// TwinCAT 3 PLC project PIDtanklevel
// ProgramVersion: 3.1.4024.12
// libraries:
//   Tc2_ControllerToolbox, * (Beckhoff Automation GmbH)
//   Tc2_ModbusSrv, * (Beckhoff Automation GmbH)
//   Tc2_Standard, * (Beckhoff Automation GmbH)
//   Tc2_System, * (Beckhoff Automation GmbH)
//   Tc3_Module, * (Beckhoff Automation GmbH)
// project tree:
//   GVLs/ GlobalTags.TcGVL, InputOutputArea.TcGVL
//   / PlcTask.TcTTO
//   POUs/ ElectricBox.TcPOU, InputOutputConvert.TcPOU, MAIN.TcPOU, ModbusRead.TcPOU, ModbusWrite.TcPOU, PID.TcPOU

CONFIGURATION PIDtanklevel
    RESOURCE PLC ON TwinCAT3
        TASK PlcTask(INTERVAL := T#10ms, PRIORITY := 20);
        PROGRAM MAIN WITH PlcTask : MAIN;
    END_RESOURCE
END_CONFIGURATION

// ---- GVLs/GlobalTags.TcGVL
VAR_GLOBAL
	//
	Start 			: BOOL;
	Reset 			: BOOL;
	Stop  			: BOOL;
	//
	StartLight		: BOOL;
	ResetLight		: BOOL;
	StopLight		: BOOL;
	//
	LevelMeter 		: INT;
	FlowMeter		: INT;
	SetPoint		: INT;
	//
	FillValve		: INT;
	DischargeValve	: INT;
	SP				: INT;
	PV				: INT;
	//
	SystemStarted	: BOOL;
END_VAR

// ---- GVLs/InputOutputArea.TcGVL
VAR_GLOBAL
	InputBitArea 		: ARRAY[0..1] OF BYTE;
	OutputBitArea 		: ARRAY[0..1] OF BYTE;
	
	InputWordArea		: ARRAY[0..2] OF WORD;
	OutputWordArea		: ARRAY[0..3] OF WORD;
END_VAR

// ---- POUs/MAIN.TcPOU
PROGRAM MAIN
VAR
	InputOutputConvert: InputOutputConvert;
	PID: PID;
	ElectricBox: ElectricBox;
END_VAR

ModbusRead();
ModbusWrite();
InputOutputConvert();
PID();
ElectricBox();

END_PROGRAM

// ---- POUs/InputOutputConvert.TcPOU
FUNCTION_BLOCK InputOutputConvert
VAR_INPUT
END_VAR
VAR_OUTPUT
END_VAR
VAR
END_VAR


//Inputs
LevelMeter := (WORD_TO_INT(InputWordArea[0])*300)/1000;
FlowMeter  := (WORD_TO_INT(InputWordArea[1])*300)/1000;
SetPoint   := (WORD_TO_INT(InputWordArea[2])*300)/1000;
//Outputs
OutputWordArea[0] := INT_TO_WORD(FillValve);
OutputWordArea[1] := INT_TO_WORD(DischargeValve);
SP		   := SetPoint;
OutputWordArea[2] := INT_TO_WORD(SP);
PV		   := LevelMeter;
OutputWordArea[3] := INT_TO_WORD(PV);

//
Start := InputBitArea[0].0;
Reset := InputBitArea[0].1;
Stop  := InputBitArea[0].2;
//
OutputBitArea[0].0 := StartLight;
OutputBitArea[0].1 := ResetLight;
OutputBitArea[0].2 := StopLight;

END_FUNCTION_BLOCK

// ---- POUs/PID.TcPOU
FUNCTION_BLOCK PID
VAR_INPUT
END_VAR
VAR_OUTPUT
END_VAR
VAR
	FB_CTRL_PID: FB_CTRL_PID;
	stCTRL_PID_PARAMS: ST_CTRL_PID_PARAMS;
	Init : BOOL:=TRUE;
	fManSyncValue : LREAL;
	fOut : LREAL;
	fState : LREAL;
	fErrId : LREAL;
	bErr   : BOOL;
	fCTRL_Mode : E_CTRL_MODE;
END_VAR


IF Init THEN
	stCTRL_PID_PARAMS.tCtrlCycleTime 	:= T#10MS;
	stCTRL_PID_PARAMS.tTaskCycleTime 	:= T#10MS;
	stCTRL_PID_PARAMS.fKp				:= 15.0;
	stCTRL_PID_PARAMS.tTn				:= T#20S;
	stCTRL_PID_PARAMS.tTv				:= T#0S;
	stCTRL_PID_PARAMS.tTd				:= T#0S;
	stCTRL_PID_PARAMS.fOutMaxLimit		:= 1000;
	stCTRL_PID_PARAMS.fOutMinLimit		:= -1000;
	stCTRL_PID_PARAMS.bPInTheFeedbackPath := TRUE;
	stCTRL_PID_PARAMS.bDInTheFeedbackPath := TRUE;
	
	Init := FALSE;
END_IF

IF NOT SystemStarted THEN
	fCTRL_Mode := eCTRL_MODE_PASSIVE;
ELSE
	fCTRL_Mode := eCTRL_MODE_ACTIVE;	
END_IF

IF Reset THEN
	fCTRL_Mode := eCTRL_MODE_RESET;
END_IF

FB_CTRL_PID(
	fSetpointValue:= INT_TO_LREAL(SetPoint), 
	fActualValue:= INT_TO_LREAL(LevelMeter), 
	fManSyncValue:= fManSyncValue, 
	bSync:= FALSE, 
	eMode:= fCTRL_Mode, 
	bHold:= FALSE, 
	fOut=> fOut, 
	bARWactive=> , 
	eState=> fState, 
	eErrorId=> fErrId, 
	bError=> bErr, 
	stParams:= stCTRL_PID_PARAMS);
	
IF fOut >= 0 THEN
	FillValve := LREAL_TO_INT(fOut);
	DischargeValve := 0;
ELSE
	FillValve := 0;
	DischargeValve := ABS(LREAL_TO_INT(fOut));
END_IF

END_FUNCTION_BLOCK

// ---- POUs/ElectricBox.TcPOU
FUNCTION_BLOCK ElectricBox
VAR_INPUT
END_VAR
VAR_OUTPUT
END_VAR
VAR
END_VAR

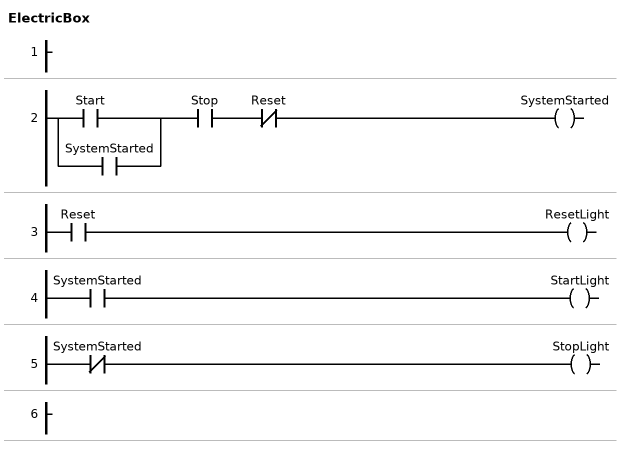
// NETWORK 1

// NETWORK 2
SystemStarted := (Start OR SystemStarted) AND Stop AND NOT Reset;

// NETWORK 3
ResetLight := Reset;

// NETWORK 4
StartLight := SystemStarted;

// NETWORK 5
StopLight := NOT SystemStarted;

// NETWORK 6

END_FUNCTION_BLOCK

// ---- POUs/ModbusRead.TcPOU
PROGRAM ModbusRead
VAR
	FB_MBReadInputs: FB_MBReadInputs;
	tReadInput: TON;
	bReadExecute: BOOL;
	
	IP 		: STRING:='127.0.0.1';
	Port 	: UINT:=505;
	ID 		: BYTE:=255;
	
	FB_MBReadInputRegs: FB_MBReadInputRegs;
	TON: TON;
	bInReg: BOOL;
END_VAR


tReadInput(IN:= NOT FB_MBReadInputs.bBusy, PT:=T#10MS , Q=>bReadExecute , ET=> );

FB_MBReadInputs(
	sIPAddr:= IP, 
	nTCPPort:= Port, 
	nUnitID:= ID, 
	nQuantity:= 16, 
	nMBAddr:= 0, 
	cbLength:= SIZEOF(InputBitArea), 
	pDestAddr:= ADR(InputBitArea), 
	bExecute:= bReadExecute, 
	tTimeout:= T#1S, 
	bBusy=> , 
	bError=> , 
	nErrId=> , 
	cbRead=> );

TON(IN:= NOT FB_MBReadInputRegs.bBusy , PT:=T#10MS , Q=>bInReg , ET=> );
	
FB_MBReadInputRegs(
	sIPAddr:= IP, 
	nTCPPort:= Port, 
	nUnitID:= ID, 
	nQuantity:= 3, 
	nMBAddr:= 0, 
	cbLength:= SIZEOF(InputWordArea), 
	pDestAddr:= ADR(InputWordArea), 
	bExecute:= bInReg, 
	tTimeout:= T#1S, 
	bBusy=> , 
	bError=> , 
	nErrId=> , 
	cbRead=> );

END_PROGRAM

// ---- POUs/ModbusWrite.TcPOU
PROGRAM ModbusWrite
VAR
	FB_MBWriteCoils: FB_MBWriteCoils;
	tExecute: TON;
	bExecute: BOOL;
	
	IP 		: STRING:='127.0.0.1';
	Port 	: UINT:=505;
	ID 		: BYTE:=255;
	
	FB_MBWriteRegs: FB_MBWriteRegs;
	TON: TON;
	bWriteReg: BOOL;
END_VAR


tExecute(IN:= NOT FB_MBWriteCoils.bBusy, PT:= T#10MS, Q=> bExecute, ET=> );

FB_MBWriteCoils(
	sIPAddr:= IP, 
	nTCPPort:= Port, 
	nUnitID:= ID, 
	nQuantity:= 16, 
	nMBAddr:= 0, 
	cbLength:= SIZEOF(OutputBitArea), 
	pSrcAddr:= ADR(OutputBitArea), 
	bExecute:= bExecute, 
	tTimeout:= T#1S, 
	bBusy=> , 
	bError=> , 
	nErrId=> );
	
TON(IN:= NOT FB_MBWriteRegs.bBusy, PT:= T#10MS, Q=> bWriteReg, ET=> );
	
FB_MBWriteRegs(
	sIPAddr:= IP, 
	nTCPPort:= Port, 
	nUnitID:= ID, 
	nQuantity:= 4, 
	nMBAddr:= 0, 
	cbLength:= SIZEOF(OutputWordArea), 
	pSrcAddr:= ADR(OutputWordArea), 
	bExecute:= bWriteReg, 
	tTimeout:= T#1S, 
	bBusy=> , 
	bError=> , 
	nErrId=> );

END_PROGRAM
